PROGRAM MAIN
VAR
	a : ARRAY[0..5] OF REAL;
	b : ARRAY[10..15] OF REAL;
END_VAR


ListOfINTTest();
ListTest();
WrappableListExample();

QuickSortTest();
SortTest();
ComparisonTest();

END_PROGRAM

(* stored: Version 1.1.0.1, ProductVersion 3.1.4024.11
   POU MAIN: Id {1a83c779-8278-4247-a37a-c1c0cf8a1ae2}, SpecialFunc None *)
